// TIA Portal V19 export
TYPE "Peeler_Status"
   STRUCT
      Lift : "ValveMachine_COut";
      Extension : "ValveMachine_COut";
      Is_Up : Bool;
      Is_Dwn : Bool;
   END_STRUCT;
END_TYPE
